TYPE TcaLaserDistanceSenorService :
STRUCT

END_STRUCT
END_TYPE

(* stored: Version 1.1.0.1
   DUT TcaLaserDistanceSenorService: Id {46cef554-d0a4-4910-a7f6-ce08ec21fecf} *)
